FUNCTION_BLOCK PWM_Output
VAR_INPUT
END_VAR
VAR_OUTPUT
END_VAR
VAR
END_VAR

END_FUNCTION_BLOCK

(* stored: Version 1.1.0.1, ProductVersion 3.1.4022.18
   POU PWM_Output: Id {563ecf95-0183-4061-b981-aa77c1abbdf1}, SpecialFunc None *)
